Yaskawa INFORM job: R1_W35-36-A1(90,180)KM-OK.JBI

/JOB
//NAME R1_W35-36-A1(90,180)KM-OK
///FOLDERNAME KRIS-SCIANA
//POS
///NPOS 69,69,0,4,0,0
///TOOL 0
///POSTYPE PULSE
///PULSE
C00000=-33428,-25345,-55167,-52708,57910,80446
C00001=-40351,-26041,-45976,-52269,50402,81397
C00002=-41423,-24843,-44302,-51927,49554,81305
C00003=-42396,-23590,-43414,-51294,49084,80996
C00004=-41423,-24843,-44302,-51927,49554,81305
C00005=-52197,-28047,-55915,-20249,51078,73361
C00006=-52201,-28312,-55298,-20389,50592,73462
C00007=-52197,-28047,-55915,-20249,51078,73361
C00008=-51548,-29426,-58034,-20595,51789,73486
C00009=-49863,-32773,-63230,-21494,53574,73803
C00010=-115393,-121918,-105566,22441,32434,54566
C00011=-115738,-112266,-99473,22119,33651,54745
C00012=-115865,-108673,-97058,22055,34020,54783
C00013=-115984,-105187,-95822,21624,35012,55021
C00014=-115865,-108673,-97058,22055,34020,54783
C00015=-100189,-107189,-96672,-13796,34365,69400
C00016=-100201,-106907,-95572,-13970,33846,69495
C00017=-100189,-107189,-96672,-13796,34365,69400
C00018=-99280,-110350,-98933,-14890,34300,69965
C00019=-96833,-118682,-104605,-17912,34032,71535
C00020=-105118,-108011,-113982,7982,53975,63605
C00021=-88402,-93309,-101613,-4021,53517,70303
C00022=-85657,-86027,-96738,-5932,54420,71360
C00023=-85657,-86238,-95900,-5976,53800,71395
C00024=-85657,-86027,-96738,-5932,54420,71360
C00025=-88898,-98629,-94424,-9032,36755,70744
C00026=-89964,-93987,-92056,-7719,37565,70068
C00027=-90400,-92057,-91281,-7177,38034,69788
C00028=-89774,-94840,-92698,-7928,37542,70175
C00029=-72922,-111787,-110466,-23490,42948,78042
C00030=-76129,-94799,-105626,10324,50692,61184
C00031=-80813,-78516,-88866,31374,50295,50464
C00032=-85919,-63473,-69401,51740,53305,41731
C00033=-85689,-63252,-68410,51919,52861,41570
C00034=-84470,-62123,-67823,51201,52325,41987
C00035=-85689,-63252,-68410,51919,52861,41570
C00036=-92588,-72655,-82010,53195,58926,41392
C00037=-73945,-95291,-113067,15746,66917,59956
C00038=-58434,-55891,-99783,-5213,90279,77372
C00039=-58848,-54858,-92727,-5051,86459,77405
C00040=-82964,-50529,-90185,4565,87055,70314
C00041=-82850,-46991,-92810,4524,90473,70471
C00042=-69976,-56638,-96571,9667,87584,76933
C00043=-71132,-55955,-92565,10137,85620,76434
C00044=-45687,-51668,-90195,-272,84985,83971
C00045=-45786,-48647,-92419,-232,87906,83936
C00046=-37246,-33085,-86176,-12581,97104,85034
C00047=-20453,-14794,-67982,-36579,105452,88184
C00048=-18131,2025,-47947,-44636,114275,84011
C00049=-23953,4875,-45887,-42681,111998,82975
C00050=-27421,-11418,-68052,-34880,104542,86047
C00051=-66885,-28498,-82158,-7865,97243,66261
C00052=-67654,-32939,-80739,-7533,94057,66244
C00053=-89648,-24444,-75126,388,94146,60009
C00054=-85856,-26926,-82512,-1000,97425,61051
C00055=-54513,-24720,-66467,-20016,74026,58804
C00056=-56472,-22787,-62043,-19135,71978,58501
C00057=-57155,-21140,-60033,-18803,71466,58359
C00058=-56423,-23526,-61352,-19244,71226,58641
C00059=-57225,-21245,-61020,-18713,71977,58251
C00060=-58027,-19371,-60210,-18283,74444,57552
C00061=-57914,-19492,-60492,-18334,74571,57569
C00062=-56844,-20676,-59861,-18960,71654,58430
C00063=-56490,-22635,-62151,-19111,72111,58473
C00064=-54532,-24553,-66568,-19992,74162,58775
C00065=-48154,-122345,-116911,-19991,54442,58776
C00066=-113071,-122345,-116911,-19991,54442,58776
C00067=-113071,-122345,-116911,-19991,54442,58776
C00068=3488,-122345,-116911,-19991,54442,58776
BC00000=35461,15,1075175
BC00001=35461,15,1075175
BC00002=35461,15,1075175
BC00003=35461,15,1075175
BC00004=35461,15,1075175
BC00005=35461,15,1075175
BC00006=35461,15,1075175
BC00007=35461,15,1075175
BC00008=35461,15,1075175
BC00009=35461,15,1075175
BC00010=145748,15,1075175
BC00011=145748,15,1075175
BC00012=145748,15,1075175
BC00013=145748,15,1075175
BC00014=145748,15,1075175
BC00015=145748,15,1075175
BC00016=145748,15,1075175
BC00017=145748,15,1075175
BC00018=145748,15,1075175
BC00019=145748,15,1075175
BC00020=145748,15,1075175
BC00021=145748,15,1075175
BC00022=145748,15,1075175
BC00023=145748,15,1075175
BC00024=145748,15,1075175
BC00025=145748,15,1075175
BC00026=145748,15,1075175
BC00027=145748,15,1075175
BC00028=145748,15,1075175
BC00029=145748,15,1075175
BC00030=145748,15,1075175
BC00031=145748,15,1075175
BC00032=145748,15,1075175
BC00033=145748,15,1075175
BC00034=145748,15,1075175
BC00035=145748,15,1075175
BC00036=145748,15,1075175
BC00037=144195,15,1075175
BC00038=142512,15,1075175
BC00039=142512,15,1075175
BC00040=142512,15,1075175
BC00041=142512,15,1075175
BC00042=142512,15,1075175
BC00043=142512,15,1075175
BC00044=142512,15,1075175
BC00045=142512,15,1075175
BC00046=142512,15,1075175
BC00047=142512,15,1075175
BC00048=142512,15,1075175
BC00049=142512,15,1075175
BC00050=142512,15,1075175
BC00051=127026,15,1075175
BC00052=127026,15,1075174
BC00053=127026,15,1075175
BC00054=127026,15,1075175
BC00055=70012,15,1075175
BC00056=69283,15,1075175
BC00057=68991,15,1075175
BC00058=68991,15,1075175
BC00059=68991,15,1075175
BC00060=58055,15,1075175
BC00061=54728,15,1075175
BC00062=19619,15,1075175
BC00063=19910,15,1075175
BC00064=20639,15,1075175
BC00065=20639,15,1075174
BC00066=20639,15,1075174
BC00067=20639,521461,1075174
BC00068=21569,521461,1075174
///POSTYPE BASE
///RECTAN
///RCONF 0,0,0,0,1,0,0,0,0,0,0,0,0,0,0,0,0,0,0,0,0,0,0,0
P00006=2.006,1.622,-0.565,0.0000,0.0000,0.0000
P00021=0.073,2.058,-0.109,0.0000,0.0000,0.0000
P00022=2.006,1.622,-0.565,0.0000,0.0000,0.0000
///RCONF 0,0,0,0,0,0,0,0,0,0,0,0,0,0,0,0,0,0,0,0,0,0,0,0
P00030=-0.014,-0.768,0.131,0.0000,0.0000,0.0000
//INST
///DATE 2024/12/27 11:40
///ATTR SC,RW
///GROUP1 RB1,BS1
NOP
'r1_W35-36-A1(90,180)
'Path S1030 (for W465)
SFTOF
MOVJ C00000 BC00000 VJ=10.00
MOVJ C00001 BC00001 VJ=20.00
MOVL C00002 BC00002 V=60.0
REFP 3 C00003 BC00003
CALL JOB:SEARCH-R1
SET P021 P006
SFTON P021
MOVL C00004 BC00004 V=60.0
MOVL C00005 BC00005 V=60.0
REFP 3 C00006 BC00006
CALL JOB:SEARCH-R1
SET P021 P006
SFTON P021
MOVL C00007 BC00007 V=60.0
MOVL C00008 BC00008 V=166.7
MOVL C00009 BC00009 V=166.7
'Path S1031 (for W465)
SFTOF
MOVL C00010 BC00010 V=166.7
MOVL C00011 BC00011 V=166.7
MOVL C00012 BC00012 V=60.0
REFP 3 C00013 BC00013
CALL JOB:SEARCH-R1
SET P022 P006
SFTON P022
MOVL C00014 BC00014 V=60.0
MOVL C00015 BC00015 V=60.0
REFP 3 C00016 BC00016
CALL JOB:SEARCH-R1
SET P022 P006
SFTON P022
MOVL C00017 BC00017 V=60.0
MOVL C00018 BC00018 V=166.7
MOVL C00019 BC00019 V=166.7
'Path VIA1148
SFTOF
MOVJ C00020 BC00020 VJ=20.00
MOVJ C00021 BC00021 VJ=10.00
MOVL C00022 BC00022 V=83.3
REFP 3 C00023 BC00023
CALL JOB:SEARCH-R1
SET P030 P006
SFTON P030
MOVL C00024 BC00024 V=83.3
MOVJ C00025 BC00025 VJ=10.00
MOVL C00026 BC00026 V=66.7
REFP 3 C00027 BC00027
CALL JOB:SEARCH-R1
SET P030 P006
SFTON P030
MOVL C00028 BC00028 V=83.3
MOVJ C00029 BC00029 VJ=50.00
MOVJ C00030 BC00030 VJ=50.00
MOVJ C00031 BC00031 VJ=50.00
MOVJ C00032 BC00032 VJ=50.00
MOVL C00033 BC00033 V=66.7
REFP 3 C00034 BC00034
CALL JOB:SEARCH-R1
SET P030 P006
SFTON P030
MOVL C00035 BC00035 V=83.3
MOVJ C00036 BC00036 VJ=50.00
MOVJ C00037 BC00037 VJ=50.00
SFTOF
MOVJ C00038 BC00038 VJ=10.00
SFTON P030
MACRO1 MJ#(0) ARGF7
MOVJ C00039 BC00039 VJ=10.00
ARCON
MOVL C00040 BC00040 V=11.7
ARCOF
MOVJ C00041 BC00041 VJ=10.00
MOVJ C00042 BC00042 VJ=60.00
MOVJ C00043 BC00043 VJ=10.00
ARCON
MOVL C00044 BC00044 V=11.7
ARCOF
MOVJ C00045 BC00045 VJ=10.00
MOVJ C00046 BC00046 VJ=10.00
MOVJ C00047 BC00047 VJ=10.00
MACRO1 MJ#(0) ARGF6
MOVJ C00048 BC00048 VJ=10.00
MOVL C00049 BC00049 V=11.7
ARCOF
MOVJ C00050 BC00050 VJ=10.00
MOVJ C00051 BC00051 VJ=20.00
MACRO1 MJ#(0) ARGF7
MOVJ C00052 BC00052 VJ=10.00
ARCON
MOVL C00053 BC00053 V=11.7
ARCOF
MOVJ C00054 BC00054 VJ=10.00
'Path W1032
SFTOF
SFTON P022
MOVJ C00055 BC00055 VJ=20.00
MOVJ C00056 BC00056 VJ=20.00
MOVL C00057 BC00057 V=100.0 PL=0
REFP 1 C00058 BC00058
REFP 2 C00059 BC00059
MACRO1 MJ#(0) ARGF7
ARCON
MOVL C00060 BC00060 V=7.5
SFTON P021
MOVL C00061 BC00061 V=7.5
MOVL C00062 BC00062 V=7.5
ARCOF
MOVL C00063 BC00063 V=166.7
MOVL C00064 BC00064 V=250.0
SFTOF
MOVJ C00065 BC00065 VJ=80.00
COMM MOVJ C00066 BC00066 VJ=100.00
COMM MOVJ C00067 BC00067 VJ=100.00
COMM MOVJ C00068 BC00068 VJ=100.00
END
